FUNCTION_BLOCK FB_TimerPulse

VAR
	fbTP : TP := (PT := T#10S);
	bResult : BOOL;
	bOn : BOOL;
END_VAR


fbTP(IN := bOn);
IF fbTP.Q THEN
	bResult := TRUE;
ELSE
	bResult  := FALSE;
END_IF

END_FUNCTION_BLOCK

(* stored: Version 1.1.0.1, ProductVersion 3.1.4024.16
   POU FB_TimerPulse: Id {85e6696d-91c5-4d02-8cea-3e8819717505}, SpecialFunc None *)
